FUNCTION_BLOCK ORDER_1D_MOVETO_PARALLEL_PLANE (* 1D_MOVETO_PARALLEL_PLANE with FILE_WRITER inside *)
  (* Standard: 61499-2 *)
  (* Version 1.0, 10-05-12, GASR, Universidade do Estado de Santa Catarina *)
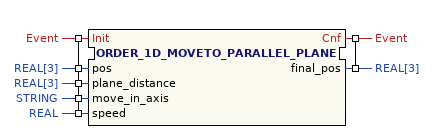
  EVENT_INPUT
    Init WITH pos, plane_distance, move_in_axis, speed;
  END_EVENT
  EVENT_OUTPUT
    Cnf WITH final_pos;
  END_EVENT
  VAR_INPUT
    pos : ARRAY [0..2] OF REAL; (* Machine position *)
    plane_distance : ARRAY [0..2] OF REAL; (* Security plane position *)
    move_in_axis : STRING; (* 'x', 'y' or 'z' *)
    speed : REAL := 0; (* Feedrate in m/s *)
  END_VAR
  VAR_OUTPUT
    final_pos : ARRAY [0..2] OF REAL; (* Final position *)
  END_VAR
  FBS
    1d_moveto_parallel_plane : 1D_MOVETO_PARALLEL_PLANE;
    order_1d_moveto_parallel_plane : FILE_WRITER_7_LINEAR_MOVE;
  END_FBS
  EVENT_CONNECTIONS
    1d_moveto_parallel_plane.Send TO order_1d_moveto_parallel_plane.REQ;
    1d_moveto_parallel_plane.Cnf TO Cnf;
    order_1d_moveto_parallel_plane.RSP TO 1d_moveto_parallel_plane.Req;
    Init TO 1d_moveto_parallel_plane.Init;
  END_CONNECTIONS
  DATA_CONNECTIONS
    1d_moveto_parallel_plane.final_pos TO final_pos;
    1d_moveto_parallel_plane.final_pos TO out_pos;
    1d_moveto_parallel_plane.v_coef TO order_1d_moveto_parallel_plane.P7;
    1d_moveto_parallel_plane.out_speed TO order_1d_moveto_parallel_plane.P6;
    1d_moveto_parallel_plane.final_pos TO order_1d_moveto_parallel_plane.P5;
    1d_moveto_parallel_plane.t0 TO order_1d_moveto_parallel_plane.P4;
    1d_moveto_parallel_plane.coef_b TO order_1d_moveto_parallel_plane.P2;
    1d_moveto_parallel_plane.t TO order_1d_moveto_parallel_plane.P3;
    1d_moveto_parallel_plane.eq_id TO order_1d_moveto_parallel_plane.P0;
    1d_moveto_parallel_plane.coef_a TO order_1d_moveto_parallel_plane.P1;
    plane_distance TO 1d_moveto_parallel_plane.plane_distance;
    speed TO 1d_moveto_parallel_plane.speed;
    move_in_axis TO 1d_moveto_parallel_plane.move_in_axis;
    pos TO 1d_moveto_parallel_plane.pos;
  END_CONNECTIONS
END_FUNCTION_BLOCK
